// TIA Portal project "MITOMI G2 V1.8" (V17)

(* hardware
DEVICE "S7-1500/ET200MP station_1"  S7-1500 station
   slot 0: "Rail_0"  Rack  6ES7 590-1***0-0AA0
   slot 0: "PM 70W 120/230VAC"  PM 70W 120/230VAC  6EP1332-4BA00
   slot 1: "PLC_1"  CPU 1512C-1 PN  6ES7 512-1CK01-0AB0  V2.8
      slot 3: "CPU display_1"  6ES7591-1AA00-0AA0
      slot 32768: "PROFINET interface_1"  X1
         slot 32769: "Port_1"  X1 P1
         slot 32770: "Port_2"  X1 P2
      slot 34817: "Virtual CP interface port_1"  Virtual CP interface port  Virtual CP interface port
   slot 2: "DQ 16x24VDC/0.5A HF_1"  DQ 16x24VDC/0.5A HF  6ES7 522-1BH01-0AB0  V1.1
   slot 3: "AI 8xU/I/RTD/TC ST_1"  AI 8xU/I/RTD/TC ST  6ES7 531-7KF00-0AB0  V2.2
   slot 4: "AQ 4xU/I ST_1"  AQ 4xU/I ST  6ES7 532-5HD00-0AB0  V2.2
   slot 5: "DQ 16x24VDC/0.5A ST_1"  DQ 16x24VDC/0.5A ST  6ES7 522-1BH00-0AB0  V1.0
*)

// ===== PLC "PLC_1"  CPU 1512C-1 PN =====

VAR_GLOBAL   // PLC tag table "Default tag table"
   "RTD_sensor" AT %IW40 : Int;
   "PWM_4" AT %M1.0 : Bool;
   "PWM_4_DC" AT %MD2 : Real;
   "FR_sensor1" AT %IW34 : Int;
   "FR" AT %MD8 : Real;
   "PWM_4_T" AT %MD12 : Time;
   "Pressure_actual" AT %IW32 : Int;   // 27648
   "Pressure_set" AT %QW34 : Int;   // 27648
   "Peltier-relay" AT %Q6.0 : Bool;
   "PID_enable" AT %M10.0 : Bool;
   "PID_manual_pressure" AT %MD16 : Real;
   "FR_sensor2" AT %IW36 : Int;
   "FR_sensor3" AT %IW38 : Int;
   "Timer1" AT %T10 : Timer;
   "Timer2" AT %T20 : Timer;
END_VAR

VAR_GLOBAL   // PLC tag table "Solenoid valves"
   "valve0_0" AT %Q0.0 : Bool;
   "valve0_1" AT %Q0.1 : Bool;
   "valve0_2" AT %Q0.2 : Bool;
   "valve0_3" AT %Q0.3 : Bool;
   "valve0_4" AT %Q0.4 : Bool;
   "valve0_5" AT %Q0.5 : Bool;
   "valve0_6" AT %Q0.6 : Bool;
   "valve0_7" AT %Q0.7 : Bool;
   "valve1_0" AT %Q1.0 : Bool;
   "valve1_1" AT %Q1.1 : Bool;
   "valve1_2" AT %Q1.2 : Bool;
   "valve1_3" AT %Q1.3 : Bool;
   "valve1_4" AT %Q1.4 : Bool;
   "valve1_5" AT %Q1.5 : Bool;
   "valve1_6" AT %Q1.6 : Bool;
   "valve1_7" AT %Q1.7 : Bool;
   "valve2_0" AT %Q2.0 : Bool;
   "valve2_1" AT %Q2.1 : Bool;
   "valve2_2" AT %Q2.2 : Bool;
   "valve2_3" AT %Q2.3 : Bool;
   "valve2_4" AT %Q2.4 : Bool;
   "valve2_5" AT %Q2.5 : Bool;
   "valve2_6" AT %Q2.6 : Bool;
   "valve2_7" AT %Q2.7 : Bool;
   "valve3_0" AT %Q3.0 : Bool;
   "valve3_1" AT %Q3.1 : Bool;
   "valve3_2" AT %Q3.2 : Bool;
   "valve3_3" AT %Q3.3 : Bool;
   "valve3_4" AT %Q3.4 : Bool;
   "valve3_5" AT %Q3.5 : Bool;
   "valve3_6" AT %Q3.6 : Bool;
   "valve3_7" AT %Q3.7 : Bool;
   "valve4_0" AT %Q4.0 : Bool;
   "valve4_1" AT %Q4.1 : Bool;
   "valve4_2" AT %Q4.2 : Bool;
   "valve4_3" AT %Q4.3 : Bool;
   "valve4_4" AT %Q4.4 : Bool;
   "valve4_5" AT %Q4.5 : Bool;
   "valve4_6" AT %Q4.6 : Bool;
   "valve4_7" AT %Q4.7 : Bool;
   "valve5_0" AT %Q5.0 : Bool;
   "valve5_1" AT %Q5.1 : Bool;
   "valve5_2" AT %Q5.2 : Bool;
   "valve5_3" AT %Q5.3 : Bool;
   "valve5_4" AT %Q5.4 : Bool;
   "valve5_5" AT %Q5.5 : Bool;
   "valve5_6" AT %Q5.6 : Bool;
   "valve5_7" AT %Q5.7 : Bool;
   "valve6_0" AT %Q7.0 : Bool;
   "valve6_1" AT %Q7.1 : Bool;
   "valve6_2" AT %Q7.2 : Bool;
   "valve6_3" AT %Q7.3 : Bool;
END_VAR

VAR_GLOBAL   // PLC tag table "PMW_tags"
   "pwm_1_ctrl" AT %Q512.0 : "type_PWM_control";
   "pwm_2_ctrl" AT %Q524.0 : "type_PWM_control";
   "pwm_3_ctrl" AT %Q536.0 : "type_PWM_control";
   "pwm_4_ctrl" AT %Q548.0 : "type_PWM_control";
   "pwm_12_odd" AT %M0.6 : Bool;
   "pwm_34_odd" AT %M0.7 : Bool;
   "pwm_12_f1" AT %M0.4 : Bool;
   "pwm_12_f2" AT %M0.5 : Bool;
   "time_temp1" AT %MD41 : Time;
   "time_temp1_s5t" AT %MW46 : S5Time;
END_VAR

TYPE "type_PWM_control"
   STRUCT
      Spare1 : Word;
      Duty_cycle : Int := 5000;
      Slot1 : UDInt := 2000000;
      LD_SLOT1 : Bool := true;
      LD_SLOT2 : Bool;
      LD_SLOT3 : Bool;
      LD_SLOT4 : Bool;
      MODE_SLOT : Bool;
      S2Res1 : Bool;
      S2Res2 : Bool;
      S3Res3 : Bool;
      SW_ENABLE : Bool := true;
      TM_CTRL_DQ : Bool := true;
      B9Res1 : Bool;
      SET_DQA : Bool;
      B9Res2 : Bool;
      B9Res3 : Bool;
      B9Res4 : Bool;
      B9Res5 : Bool;
      RES_ERROR : Bool;
      B10Res1 : Bool;
      B10Res2 : Bool;
      B10Res3 : Bool;
      B10Res4 : Bool;
      B10Res5 : Bool;
      B10Res6 : Bool;
      B10Res7 : Bool;
      Spare2 : Byte;
   END_STRUCT;
END_TYPE

TYPE "type_PWM_status"
   STRUCT
      ERR_PWR : Bool;
      B1Res1 : Bool;
      ERR_LD : Bool;
      ERR_PULSE : Bool;
      B1Res2 : Bool;
      B1Res3 : Bool;
      ERR_OUT_VAL : Bool;
      ERR_SLOT_VAL : Bool;
      B2Res1 : Bool;
      B2Res2 : Bool;
      STS_LD_SLOT : Bool;
      B2Res3 : Bool;
      STS_READY : Bool;
      STS_SW_ENABLE : Bool;
      B2Res4 : Bool;
      B2Res5 : Bool;
      STS_ENABLE : Bool;
      STS_DQA : Bool;
      B3Res1 : Bool;
      B3Res2 : Bool;
      B3Res3 : Bool;
      B3Res4 : Bool;
      B3Res5 : Bool;
      B3Res6 : Bool;
      B4Res : Byte;
   END_STRUCT;
END_TYPE

DATA_BLOCK "Solenoid valves"   // DB1
{ S7_Optimized_Access := 'TRUE' }
VERSION : 0.1
   VAR
      S00 : Bool;
      S01 : Bool;
      S02 : Bool;
      S03 : Bool;
      S04 : Bool;
      S05 : Bool;
      S06 : Bool;
      S07 : Bool;
      S10 : Bool;
      S11 : Bool;
      S12 : Bool;
      S13 : Bool;
      S14 : Bool;
      S15 : Bool;
      S16 : Bool;
      S17 : Bool;
      S20 : Bool;
      S21 : Bool;
      S22 : Bool;
      S23 : Bool;
      S24 : Bool;
      S25 : Bool;
      S26 : Bool;
      S27 : Bool;
      S30 : Bool;
      S31 : Bool;
      S32 : Bool;
      S33 : Bool;
      S34 : Bool;
      S35 : Bool;
      S36 : Bool;
      S37 : Bool;
      S40 : Bool;
      S41 : Bool;
      S42 : Bool;
      S43 : Bool;
      S44 : Bool;
      S45 : Bool;
      S46 : Bool;
      S47 : Bool;
      S50 : Bool;
      S51 : Bool;
      S52 : Bool;
      S53 : Bool;
      S54 : Bool;
      S55 : Bool;
      S56 : Bool;
      S57 : Bool;
      S60 : Bool;
      S61 : Bool;
      S62 : Bool;
      S63 : Bool;
   END_VAR
BEGIN
END_DATA_BLOCK

DATA_BLOCK "PWM values"   // DB2
{ S7_Optimized_Access := 'TRUE' }
VERSION : 0.1
   VAR
      pwm1_dc : Int := 5000;
      pwm2_dc : Int := 5000;
      pwm3_dc : Int := 5000;
      pwm4_dc : Int := 5000;
      pwm1 : Bool;
      pwm2 : Bool;
      pwm3 : Bool;
      pwm4 : Bool;
      pwm1_enable : Bool;
      pwm2_enable : Bool;
      pwm3_enable : Bool;
      pwm4_enable : Bool;
      pwm1_period : DInt := 2000000;
      pwm2_period : DInt := 2000000;
      pwm3_period : DInt := 2000000;
      pwm4_period : DInt := 2000000;
      pwm1_delay_buffer : DInt;
      pwm1_delay_update : Bool;
      pwm1_delay_diff : DInt;
      pwm1_delay_timer_update_1 : Bool;
      pwm1_delay_timer_update_2 : Bool;
      pwm1_time_dint : Time;
      pwm1_time_s5t : S5Time;
      pwm1_period_buffer : DInt := 2000000;
      pwm1_period_update : Bool;
      pwm1_period_scaling : Real;
      pwm3_delay_buffer : DInt;
      pwm3_delay_update : Bool;
      pwm3_delay_diff : DInt;
      pwm3_delay_timer_update_1 : Bool;
      pwm3_delay_timer_update_2 : Bool;
      pwm3_time_dint : Time;
      pwm3_time_s5t : S5Time;
      pwm3_period_buffer : DInt := 2000000;
      pwm3_period_update : Bool;
      pwm3_period_scaling : Real;
   END_VAR
BEGIN
END_DATA_BLOCK

DATA_BLOCK "PLC DB"   // DB3
{ S7_Optimized_Access := 'TRUE' }
VERSION : 0.1
   VAR
      Flowrate_raw_1 : Real;
      Flowrate_raw_2 : Real;
      Flowrate_raw_3 : Real;
      Pressure_read_raw : Real;
      Flowrate_1 : Real;
      Flowrate_2 : Real;
      Flowrate_3 : Real;
      Temperature_RTD : Int;
      FR_control_pressure : Real;
      FR_control_flowrate : Real := 2.5;
      Pressure_read : Real;
      Pressure_write : Real;
      FR_control_off : Bool := TRUE;
   END_VAR
BEGIN
END_DATA_BLOCK

FUNCTION "Solenoid Update" : Void   // FC1, STL
{ S7_Optimized_Access := 'TRUE' }
VERSION : 0.1
BEGIN

REGION Network 1
         A     "Solenoid valves".S00;
         =     "pwm_1_ctrl".SET_DQA;
END_REGION

REGION Network 2
         A     "Solenoid valves".S01;
         =     "valve0_1";
END_REGION

REGION Network 3
         A     "Solenoid valves".S02;
         =     "pwm_2_ctrl".SET_DQA;
END_REGION

REGION Network 4
         A     "Solenoid valves".S03;
         =     "valve0_3";
END_REGION

REGION Network 5
         A     "Solenoid valves".S04;
         =     "pwm_3_ctrl".SET_DQA;
END_REGION

REGION Network 6
         A     "Solenoid valves".S05;
         =     "valve0_5";
END_REGION

REGION Network 7: DQ0.6 Suppressed for PWM
         A     "Solenoid valves".S06;
         =     "pwm_4_ctrl".SET_DQA;
END_REGION

REGION Network 8: DQ0.7 Suppressed for PWM
         A     "Solenoid valves".S07;
         =     "valve0_7";
END_REGION

REGION Network 9
         A     "Solenoid valves".S10;
         =     "valve1_0";
END_REGION

REGION Network 10
         A     "Solenoid valves".S11;
         =     "valve1_1";
END_REGION

REGION Network 11
         A     "Solenoid valves".S12;
         =     "valve1_2";
END_REGION

REGION Network 12
         A     "Solenoid valves".S13;
         =     "valve1_3";
END_REGION

REGION Network 13
         A     "Solenoid valves".S14;
         =     "valve1_4";
END_REGION

REGION Network 14
         A     "Solenoid valves".S15;
         =     "valve1_5";
END_REGION

REGION Network 15
         A     "Solenoid valves".S16;
         =     "valve1_6";
END_REGION

REGION Network 16
         A     "Solenoid valves".S17;
         =     "valve1_7";
END_REGION

REGION Network 17
         A     "Solenoid valves".S20;
         =     "valve2_0";
END_REGION

REGION Network 18
         A     "Solenoid valves".S21;
         =     "valve2_1";
END_REGION

REGION Network 19
         A     "Solenoid valves".S22;
         =     "valve2_2";
END_REGION

REGION Network 20
         A     "Solenoid valves".S23;
         =     "valve2_3";
END_REGION

REGION Network 21
         A     "Solenoid valves".S24;
         =     "valve2_4";
END_REGION

REGION Network 22
         A     "Solenoid valves".S25;
         =     "valve2_5";
END_REGION

REGION Network 23
         A     "Solenoid valves".S26;
         =     "valve2_6";
END_REGION

REGION Network 24
         A     "Solenoid valves".S27;
         =     "valve2_7";
END_REGION

REGION Network 25
         A     "Solenoid valves".S30;
         =     "valve3_0";
END_REGION

REGION Network 26
         A     "Solenoid valves".S31;
         =     "valve3_1";
END_REGION

REGION Network 27
         A     "Solenoid valves".S32;
         =     "valve3_2";
END_REGION

REGION Network 28
         A     "Solenoid valves".S33;
         =     "valve3_3";
END_REGION

REGION Network 29
         A     "Solenoid valves".S34;
         =     "valve3_4";
END_REGION

REGION Network 30
         A     "Solenoid valves".S35;
         =     "valve3_5";
END_REGION

REGION Network 31
         A     "Solenoid valves".S36;
         =     "valve3_6";
END_REGION

REGION Network 32
         A     "Solenoid valves".S37;
         =     "valve3_7";
END_REGION

REGION Network 33
         A     "Solenoid valves".S40;
         =     "valve4_0";
END_REGION

REGION Network 34
         A     "Solenoid valves".S41;
         =     "valve4_1";
END_REGION

REGION Network 35
         A     "Solenoid valves".S42;
         =     "valve4_2";
END_REGION

REGION Network 36
         A     "Solenoid valves".S43;
         =     "valve4_3";
END_REGION

REGION Network 37
         A     "Solenoid valves".S44;
         =     "valve4_4";
END_REGION

REGION Network 38
         A     "Solenoid valves".S45;
         =     "valve4_5";
END_REGION

REGION Network 39
         A     "Solenoid valves".S46;
         =     "valve4_6";
END_REGION

REGION Network 40
         A     "Solenoid valves".S47;
         =     "valve4_7";
END_REGION

REGION Network 41
         A     "Solenoid valves".S50;
         =     "valve5_0";
END_REGION

REGION Network 42
         A     "Solenoid valves".S51;
         =     "valve5_1";
END_REGION

REGION Network 43
         A     "Solenoid valves".S52;
         =     "valve5_2";
END_REGION

REGION Network 44
         A     "Solenoid valves".S53;
         =     "valve5_3";
END_REGION

REGION Network 45
         A     "Solenoid valves".S54;
         =     "valve5_4";
END_REGION

REGION Network 46
         A     "Solenoid valves".S55;
         =     "valve5_5";
END_REGION

REGION Network 47
         A     "Solenoid valves".S56;
         =     "valve5_6";
END_REGION

REGION Network 48
         A     "Solenoid valves".S57;
         =     "valve5_7";
END_REGION

REGION Network 49
         A     "Solenoid valves".S60;
         =     "valve6_0";
END_REGION

REGION Network 50
         A     "Solenoid valves".S61;
         =     "valve6_1";
END_REGION

REGION Network 51
         A     "Solenoid valves".S62;
         =     "valve6_2";
END_REGION

REGION Network 52
         A     "Solenoid valves".S63;
         =     "valve6_3";
END_REGION
END_FUNCTION

FUNCTION "Cooling" : Void   // FC2, LAD
{ S7_Optimized_Access := 'TRUE' }
VERSION : 0.1
BEGIN

REGION Network 1
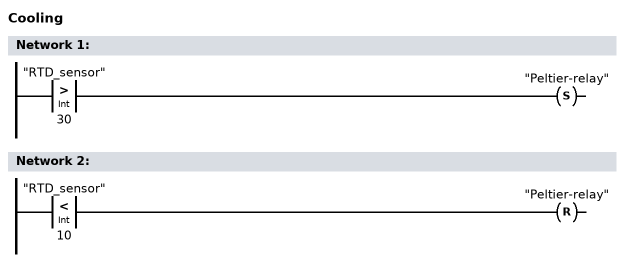
   RUNG wire#powerrail
      { S7_Templates := "SrcType := Int" } GT_Contact(in1 := "RTD_sensor", in2 := 30)
      S_Coil( "Peltier-relay" )
   END_RUNG
   // the same network as SCL:
   IF "RTD_sensor" > 30 THEN "Peltier-relay" := TRUE; END_IF;
END_REGION

REGION Network 2
   RUNG wire#powerrail
      { S7_Templates := "SrcType := Int" } LT_Contact(in1 := "RTD_sensor", in2 := 10)
      R_Coil( "Peltier-relay" )
   END_RUNG
   // the same network as SCL:
   IF "RTD_sensor" < 10 THEN "Peltier-relay" := FALSE; END_IF;
END_REGION

REGION Network 3 (STL)
         L     "RTD_sensor";
         T     "PLC DB".Temperature_RTD;
END_REGION
END_FUNCTION

FUNCTION "PWM Function" : Void   // FC4, STL
{ S7_Optimized_Access := 'TRUE' }
VERSION : 0.1
BEGIN

REGION Network 1
         A     "PWM values".pwm1_enable;
         =     "pwm_1_ctrl".TM_CTRL_DQ;
         =     "pwm_2_ctrl".TM_CTRL_DQ;
         A     "PWM values".pwm3_enable;
         =     "pwm_3_ctrl".TM_CTRL_DQ;
         =     "pwm_4_ctrl".TM_CTRL_DQ;
END_REGION

REGION Network 2
         L     "PWM values".pwm1_period;
         L     "PWM values".pwm1_period_buffer;
         <>D;
         S     "PWM values".pwm1_period_update;
   //set period update flag to true if period changes
END_REGION

REGION Network 3
         L     "PWM values".pwm3_period;
         L     "PWM values".pwm3_period_buffer;
         <>D;
         S     "PWM values".pwm3_period_update;
   //set period update flag to true if period changes
END_REGION

REGION Network 4
         A     "PWM values".pwm1_period_update;
         JCN   F1;

         L     "PWM values".pwm1_period;
         DTR;
         L     "PWM values".pwm1_period_buffer;
         DTR;
         /R;
         T     "PWM values".pwm1_period_scaling;

   // calculate scaling of period
         L     "PWM values".pwm1_delay_buffer;
         DTR;
         L     "PWM values".pwm1_period_scaling;
         *R;
         RND;
         T     "PWM values".pwm1_delay_buffer;
   // update delay to scaled delay
         L     "PWM values".pwm1_period;
         T     "PWM values".pwm1_period_buffer;
   // transfer new period to period buffer
         R     "PWM values".pwm1_period_update;
         S     "PWM values".pwm1_delay_update;
   F1:   NOP   0;
END_REGION

REGION Network 5
         A     "PWM values".pwm3_period_update;
         JCN   F2;

         L     "PWM values".pwm3_period;
         DTR;
         L     "PWM values".pwm3_period_buffer;
         DTR;
         /R;
         T     "PWM values".pwm3_period_scaling;

   // calculate scaling of period
         L     "PWM values".pwm3_delay_buffer;
         DTR;
         L     "PWM values".pwm3_period_scaling;
         *R;
         RND;
         T     "PWM values".pwm3_delay_buffer;
   // update delay to scaled delay
         L     "PWM values".pwm3_period;
         T     "PWM values".pwm3_period_buffer;
   // transfer new period to period buffer
         R     "PWM values".pwm3_period_update;
         S     "PWM values".pwm3_delay_update;
   F2:   NOP   0;
END_REGION

REGION Network 6
         L     "PWM values".pwm1_period;
         L     10000;
         /D;
         L     "PWM values".pwm1_dc;
         ITD;
         *D;
         L     1000;
         /D;
         L     "PWM values".pwm1_delay_buffer;
         <>D;
         S     "PWM values".pwm1_delay_update;
   // compare the current desired delay with buffered delay
END_REGION

REGION Network 7
         L     "PWM values".pwm3_period;
         L     10000;
         /D;
         L     "PWM values".pwm3_dc;
         ITD;
         *D;
         L     1000;
         /D;
         L     "PWM values".pwm3_delay_buffer;
         <>D;
         S     "PWM values".pwm3_delay_update;
   // compare the current desired delay with buffered delay
END_REGION

REGION Network 8
         A     "PWM values".pwm1_delay_update;
         AN(;
         O     "PWM values".pwm1_delay_timer_update_1;
         O     "PWM values".pwm1_delay_timer_update_2;
         );

         JCN   A1;
         CLR;

         L     "PWM values".pwm1_dc;
         T     "pwm_1_ctrl".Duty_cycle;
         L     10000;
         L     "PWM values".pwm1_dc;
         -I;
         T     "pwm_2_ctrl".Duty_cycle;
   //update dutycycle
         L     "PWM values".pwm1_period;
         T     "pwm_1_ctrl".Slot1;
         T     "pwm_2_ctrl".Slot1;
   //update period
         L     "PWM values".pwm1_period;
         L     10000;
         /D;
         L     "PWM values".pwm1_dc;
         ITD;
         *D;
         L     1000;
         /D;
         L     "PWM values".pwm1_delay_buffer;
         -D;
         T     "PWM values".pwm1_delay_diff;  //in ms
   // calculate difference between current delay and buffered delay

         L     "PWM values".pwm1_delay_diff;
         L     0;
         >=D;
         =     "PWM values".pwm1_delay_timer_update_2;
         NOT;
         =     "PWM values".pwm1_delay_timer_update_1;

         L     "PWM values".pwm1_delay_diff;
         DTR;
         ABS;
         RND;
         T     "PWM values".pwm1_time_dint;

         CALL  T_CONV
         ( IN  := "PWM values".pwm1_time_dint,
           OUT := "PWM values".pwm1_time_s5t  //S5 Time as output
         );

         SET;
         R     "PWM values".pwm1_delay_update;  //and reset update flag
   A1:   NOP   0;
END_REGION

REGION Network 9
         A     "PWM values".pwm3_delay_update;
         AN(;
         O     "PWM values".pwm3_delay_timer_update_1;
         O     "PWM values".pwm3_delay_timer_update_2;
         );

         JCN   A2;
         CLR;

         L     "PWM values".pwm3_dc;
         T     "pwm_3_ctrl".Duty_cycle;
         L     10000;
         L     "PWM values".pwm3_dc;
         -I;
         T     "pwm_4_ctrl".Duty_cycle;
   //update dutycycle
         L     "PWM values".pwm3_period;
         T     "pwm_3_ctrl".Slot1;
         T     "pwm_4_ctrl".Slot1;
   //update period
         L     "PWM values".pwm3_period;
         L     10000;
         /D;
         L     "PWM values".pwm3_dc;
         ITD;
         *D;
         L     1000;
         /D;
         L     "PWM values".pwm3_delay_buffer;
         -D;
         T     "PWM values".pwm3_delay_diff;  //in ms
   // calculate difference between current delay and buffered delay

         L     "PWM values".pwm3_delay_diff;
         L     0;
         >=D;
         =     "PWM values".pwm3_delay_timer_update_2;
         NOT;
         =     "PWM values".pwm3_delay_timer_update_1;

         L     "PWM values".pwm3_delay_diff;
         DTR;
         ABS;
         RND;
         T     "PWM values".pwm3_time_dint;

         CALL  T_CONV
         ( IN  := "PWM values".pwm3_time_dint,
           OUT := "PWM values".pwm3_time_s5t  //S5 Time as output
         );

         SET;
         R     "PWM values".pwm3_delay_update;  //and reset update flag
   A2:   NOP   0;
END_REGION

REGION Network 10
         A     "PWM values".pwm1_enable;
         AN    "PWM values".pwm1;
         JCN   E1;
         CLR;
         SD    "Timer1";
   E1:   NOP   0;
END_REGION

REGION Network 11
         A     "PWM values".pwm3_enable;
         AN    "PWM values".pwm3;
         JCN   E2;
         CLR;
         SD    "Timer2";
   E2:   NOP   0;
END_REGION

REGION Network 12
         A     "PWM values".pwm1_enable;
         A     "PWM values".pwm1;
         JCN   C1;  // jump end if pwm off

         A     "PWM values".pwm1_delay_timer_update_2;  //2 start later than 1
         S     "pwm_1_ctrl".SW_ENABLE;
         JC    C3;
         A     "PWM values".pwm1_delay_timer_update_1;  //1 start later than 2
         S     "pwm_2_ctrl".SW_ENABLE;
         JC    C3;
         JCN   C1;  //no update jump end
   C3:   SET;
   // jump start pwm if no delay change
         L     "PWM values".pwm1_time_s5t;
         SD    "Timer1";
   // start delay timer with difference in s5t
         A     "Timer1";
   // update pwm with timer status (1 for eclapsed and after)
         S     "pwm_2_ctrl".SW_ENABLE;
         S     "pwm_1_ctrl".SW_ENABLE;
         JCN   C1;  //jump end if timer not eclapsed

         L     "PWM values".pwm1_period;
         L     10000;
         /D;
         L     "PWM values".pwm1_dc;
         ITD;
         *D;
         L     1000;
         /D;
         T     "PWM values".pwm1_delay_buffer;  //in ms
   //elsewise set buffered delay to corrected delay
         R     "PWM values".pwm1_delay_timer_update_2;
         R     "PWM values".pwm1_delay_timer_update_1;
   C2:   SET;
         S     "pwm_1_ctrl".SW_ENABLE;
         S     "pwm_2_ctrl".SW_ENABLE;

   C1:   AN    "PWM values".pwm1;
         R     "pwm_1_ctrl".SW_ENABLE;
         R     "pwm_2_ctrl".SW_ENABLE;
END_REGION

REGION Network 13
         A     "PWM values".pwm3_enable;
         A     "PWM values".pwm3;
         JCN   G1;  // jump end if pwm off

         A     "PWM values".pwm3_delay_timer_update_2;  //2 start later than 1
         S     "pwm_3_ctrl".SW_ENABLE;
         JC    G3;
         A     "PWM values".pwm3_delay_timer_update_1;  //1 start later than 2
         S     "pwm_4_ctrl".SW_ENABLE;
         JC    G3;
         JCN   G1;  //no update jump end
   G3:   SET;
   // jump start pwm if no delay change
         L     "PWM values".pwm3_time_s5t;
         SD    "Timer2";
   // start delay timer with difference in s5t
         A     "Timer2";
   // update pwm with timer status (1 for eclapsed and after)
         S     "pwm_4_ctrl".SW_ENABLE;
         S     "pwm_3_ctrl".SW_ENABLE;
         JCN   G1;  //jump end if timer not eclapsed

         L     "PWM values".pwm3_period;
         L     10000;
         /D;
         L     "PWM values".pwm3_dc;
         ITD;
         *D;
         L     1000;
         /D;
         T     "PWM values".pwm3_delay_buffer;  //in ms
   //elsewise set buffered delay to corrected delay
         R     "PWM values".pwm3_delay_timer_update_2;
         R     "PWM values".pwm3_delay_timer_update_1;
   G2:   SET;
         S     "pwm_3_ctrl".SW_ENABLE;
         S     "pwm_4_ctrl".SW_ENABLE;

   G1:   AN    "PWM values".pwm3;
         R     "pwm_3_ctrl".SW_ENABLE;
         R     "pwm_4_ctrl".SW_ENABLE;
END_REGION
END_FUNCTION

ORGANIZATION_BLOCK "Main"   // OB1, LAD, ProgramCycle
TITLE = "Main Program Sweep (Cycle)"
{ S7_Optimized_Access := 'TRUE' }
VERSION : 0.1
   VAR_INPUT
      Initial_Call : Bool;   // Initial call of this OB
      Remanence : Bool;   // =True, if remanent data are available
   END_VAR
BEGIN

REGION Network 1
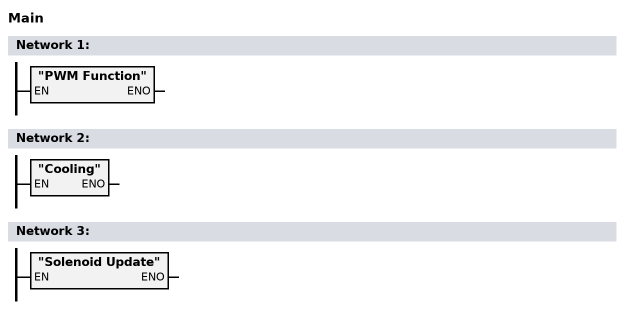
   RUNG wire#powerrail
      "PWM Function"()
   END_RUNG
   // the same network as SCL:
   "PWM Function"();
END_REGION

REGION Network 2
   RUNG wire#powerrail
      "Cooling"()
   END_RUNG
   // the same network as SCL:
   "Cooling"();
END_REGION

REGION Network 3
   RUNG wire#powerrail
      "Solenoid Update"()
   END_RUNG
   // the same network as SCL:
   "Solenoid Update"();
END_REGION
END_ORGANIZATION_BLOCK

ORGANIZATION_BLOCK "Cyclic Flowrate"   // OB30, LAD, CyclicInterrupt
{ S7_Optimized_Access := 'TRUE' }
VERSION : 0.1
   VAR_INPUT
      Initial_Call : Bool;   // Initial call of this OB
      Event_Count : Int;   // Events discarded
   END_VAR
BEGIN

REGION Network 1: Flowrate conversion
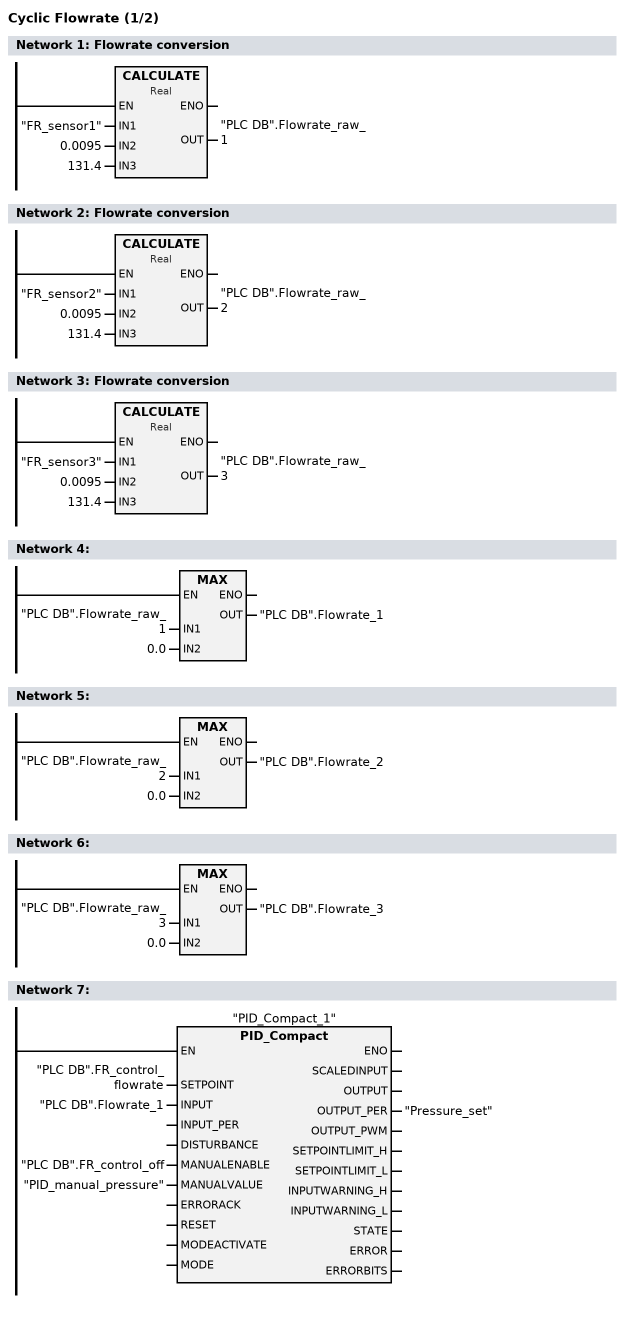
   RUNG wire#powerrail
      { S7_Templates := "SrcType := Real"; S7_Expression := "IN1*IN2-IN3" } Calculate(in1 := "FR_sensor1", in2 := 0.0095, in3 := 131.4, out => "PLC DB".Flowrate_raw_1)
   END_RUNG
   // the same network as SCL:
   "PLC DB".Flowrate_raw_1 := "FR_sensor1"*0.0095-131.4;
END_REGION

REGION Network 2: Flowrate conversion
   RUNG wire#powerrail
      { S7_Templates := "SrcType := Real"; S7_Expression := "IN1*IN2-IN3" } Calculate(in1 := "FR_sensor2", in2 := 0.0095, in3 := 131.4, out => "PLC DB".Flowrate_raw_2)
   END_RUNG
   // the same network as SCL:
   "PLC DB".Flowrate_raw_2 := "FR_sensor2"*0.0095-131.4;
END_REGION

REGION Network 3: Flowrate conversion
   RUNG wire#powerrail
      { S7_Templates := "SrcType := Real"; S7_Expression := "IN1*IN2-IN3" } Calculate(in1 := "FR_sensor3", in2 := 0.0095, in3 := 131.4, out => "PLC DB".Flowrate_raw_3)
   END_RUNG
   // the same network as SCL:
   "PLC DB".Flowrate_raw_3 := "FR_sensor3"*0.0095-131.4;
END_REGION

REGION Network 4
   "PLC DB".Flowrate_1 := MAX(IN1 := "PLC DB".Flowrate_raw_1, IN2 := 0.0);
END_REGION

REGION Network 5
   "PLC DB".Flowrate_2 := MAX(IN1 := "PLC DB".Flowrate_raw_2, IN2 := 0.0);
END_REGION

REGION Network 6
   "PLC DB".Flowrate_3 := MAX(IN1 := "PLC DB".Flowrate_raw_3, IN2 := 0.0);
END_REGION

REGION Network 7
   "PID_Compact_1"(Setpoint := "PLC DB".FR_control_flowrate,   // PID_Compact
                   Input := "PLC DB".Flowrate_1,
                   ManualEnable := "PLC DB".FR_control_off,
                   ManualValue := "PID_manual_pressure",
                   Output_PER => "Pressure_set");
END_REGION

REGION Network 8
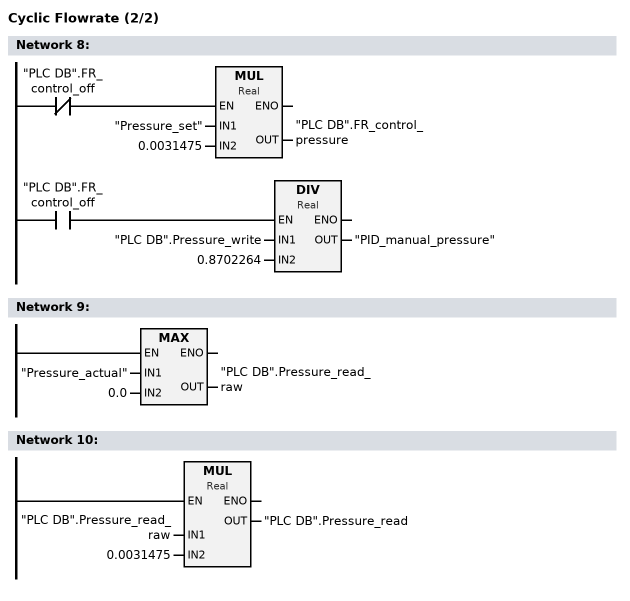
   RUNG wire#powerrail
      I_Contact( "PLC DB".FR_control_off )
      { S7_Templates := "SrcType := Real" } Mul(in1 := "Pressure_set", in2 := 0.0031475, out => "PLC DB".FR_control_pressure)
   END_RUNG
   RUNG wire#powerrail
      Contact( "PLC DB".FR_control_off )
      { S7_Templates := "SrcType := Real" } Div(in1 := "PLC DB".Pressure_write, in2 := 0.8702264, out => "PID_manual_pressure")
   END_RUNG
   // the same network as SCL:
   IF NOT "PLC DB".FR_control_off THEN "PLC DB".FR_control_pressure := "Pressure_set" * 0.0031475; END_IF;
   IF "PLC DB".FR_control_off THEN "PID_manual_pressure" := "PLC DB".Pressure_write / 0.8702264; END_IF;
END_REGION

REGION Network 9
   "PLC DB".Pressure_read_raw := MAX(IN1 := "Pressure_actual", IN2 := 0.0);
END_REGION

REGION Network 10
   RUNG wire#powerrail
      { S7_Templates := "SrcType := Real" } Mul(in1 := "PLC DB".Pressure_read_raw, in2 := 0.0031475, out => "PLC DB".Pressure_read)
   END_RUNG
   // the same network as SCL:
   "PLC DB".Pressure_read := "PLC DB".Pressure_read_raw * 0.0031475;
END_REGION
END_ORGANIZATION_BLOCK

ORGANIZATION_BLOCK "Startup"   // OB100, LAD, Startup
TITLE = "Complete Restart"
{ S7_Optimized_Access := 'TRUE' }
VERSION : 0.1
   VAR_INPUT
      LostRetentive : Bool;   // True if retentive data are lost
      LostRTC : Bool;   // True if date and time are lost
   END_VAR
BEGIN

REGION Network 1 (STL)
         SET;
         =     "pwm_1_ctrl".MODE_SLOT;
         =     "pwm_1_ctrl".LD_SLOT1;
         =     "pwm_2_ctrl".MODE_SLOT;
         =     "pwm_2_ctrl".LD_SLOT1;
         =     "pwm_3_ctrl".MODE_SLOT;
         =     "pwm_3_ctrl".LD_SLOT1;
         =     "pwm_4_ctrl".MODE_SLOT;
         =     "pwm_4_ctrl".LD_SLOT1;
         =     "pwm_12_f1";
END_REGION

REGION Network 2 (STL)
         L     2000000;
         T     "pwm_1_ctrl".Slot1;
         T     "pwm_2_ctrl".Slot1;
         T     "pwm_3_ctrl".Slot1;
         T     "pwm_4_ctrl".Slot1;
         L     5000;
         T     "pwm_1_ctrl".Duty_cycle;
         T     "pwm_2_ctrl".Duty_cycle;
         T     "pwm_3_ctrl".Duty_cycle;
         T     "pwm_4_ctrl".Duty_cycle;
END_REGION
END_ORGANIZATION_BLOCK